// SIMATIC STEP 7 (V5.x) project S7_Pro1
// CPU: CPU312(1)
// station: P_ADR_BUS
// station: Hardware
// station: SIMATIC 300 Station
// program: S7 Program(1)

SYMBOL_TABLE
"Cycle Execution"	OB 1	OB 1
END_SYMBOL_TABLE
